(* PLC project faults, TNI-Software ControlBuild 4.00.17 *)
(* stored: creationDateTime 2005-06-20T11:54:12-01:00 *)

FUNCTION_BLOCK cmd_equipment_library.faults
  VAR_INPUT  (* CB.group=Orders CB.kind=inputVars *)
    highSpeedCmd : BOOL := false;  (* CB.libelle=High speed command *)
    lowSpeedCmd : BOOL := false;  (* CB.libelle=Low speed command *)
  END_VAR
  VAR_INPUT  (* CB.group=FeedBacks CB.kind=inputVars *)
    highSpeedFB : BOOL := false;  (* CB.libelle=High speed feedback *)
    lowSpeedFB : BOOL := false;  (* CB.libelle=Low speed feedback *)
    thermalFB : BOOL := false;  (* CB.libelle=Feedback of the thermal protection of the agitator *)
  END_VAR
  VAR_INPUT  (* CB.kind=inputVars *)
    acknowledgePB : BOOL := false;  (* CB.libelle=Acknowledgement pushbutton *)
  END_VAR
  VAR_OUTPUT  (* CB.kind=outputVars *)
    generalFault : BOOL := false;  (* CB.mnemonicPatternPropertyName=grlFlt<SY><NU> CB.libelle=General fault of the agitator *)
  END_VAR
  VAR CONSTANT  (* CB.kind=parameterVars *)
    preset : DINT := 2;  (* CB.mnemonicPatternPropertyName=preset<SY><NU> CB.libelle=in seconds *)
  END_VAR
  VAR  (* CB.group=Faults CB.kind=overControlVars *)
    thermalFault : BOOL := false;  (* CB.mnemonicPatternPropertyName=thermalFlt<SY><NU> CB.libelle=Thermal (electric) fault *)
    highSpeedFBFault : BOOL := false;  (* CB.mnemonicPatternPropertyName=hSFBFlt<SY><NU> CB.libelle=High speed feedback fault *)
    lowSpeedFBFault : BOOL := false;  (* CB.mnemonicPatternPropertyName=lSFBFlt<SY><NU> CB.libelle=Low speed feedback fault *)
  END_VAR

(* LD diagram, written out as Structured Text *)
1:
IF acknowledgePB THEN thermalFault := FALSE; END_IF;
IF acknowledgePB THEN highSpeedFBFault := FALSE; END_IF;
IF acknowledgePB THEN lowSpeedFBFault := FALSE; END_IF;
IF acknowledgePB THEN generalFault := FALSE; END_IF;
2:
ton_sec_1(IN := highSpeedCmd, PT := preset);
IF ton_sec_1.Q AND NOT highSpeedFB THEN highSpeedFBFault := TRUE; END_IF;
ton_sec_2(IN := lowSpeedCmd, PT := preset);
IF ton_sec_2.Q AND NOT lowSpeedFB THEN lowSpeedFBFault := TRUE; END_IF;
3:
ton_sec_3(IN := NOT thermalFB, PT := preset);
IF ton_sec_3.Q THEN thermalFault := TRUE; END_IF;
4:
IF thermalFault OR highSpeedFBFault OR lowSpeedFBFault THEN generalFault := TRUE; END_IF;
END_FUNCTION_BLOCK
